PROGRAM MAIN

bla();

END_PROGRAM

(* stored: Version 1.1.0.1, ProductVersion 3.1.4020.6
   POU MAIN: Id {14d3af64-b01f-43e7-a2c1-878fd3bdb950}, SpecialFunc None *)
